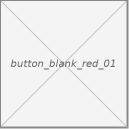
VISUALIZATION Red_Ind  // 129x129
VAR_INPUT
	m_Input_Inst : Bool;
END_VAR
    Image (0,0 127x127), invisible if: (m_Input_Inst) <> 0, image: button_blank_gray_01
    Image (0,0 127x127), invisible if: (NOT m_Input_Inst) <> 0, image: button_blank_red_01
END_VISUALIZATION

(* stored: Version 1.1.0.1, ProductVersion 3.1.4018.2
   Visu Red_Ind: Id {cca7f412-b1bc-41eb-8cea-fab03a7cecdb} *)
